FUNCTION_BLOCK OutputSender (* Composite Function Block Type *)
  (* Standard: 61499-2 *)
  (* Version 0.0, 6/20/2018, Rediska, nxtControl GmbH, template *)
  PACKAGE Main;
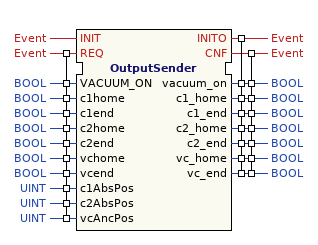
  EVENT_INPUT
    INIT; (* Initialization Request *)
    REQ WITH VACUUM_ON, c1home, c1end, c2home, c2end, vchome, vcend, c1AbsPos, c2AbsPos, vcAncPos; (* Normal Execution Request *)
  END_EVENT
  EVENT_OUTPUT
    INITO WITH vacuum_on, c1_home, c1_end, c2_home, c2_end, vc_home, vc_end; (* Initialization Confirm *)
    CNF WITH vacuum_on, c1_home, c1_end, c2_home, c2_end, vc_home, vc_end; (* Execution Confirmation *)
  END_EVENT
  VAR_INPUT
    VACUUM_ON : BOOL;
    c1home : BOOL;
    c1end : BOOL;
    c2home : BOOL;
    c2end : BOOL;
    vchome : BOOL;
    vcend : BOOL;
    c1AbsPos : UINT;
    c2AbsPos : UINT;
    vcAncPos : UINT;
  END_VAR
  VAR_OUTPUT
    vacuum_on : BOOL;
    c1_home : BOOL;
    c1_end : BOOL;
    c2_home : BOOL;
    c2_end : BOOL;
    vc_home : BOOL;
    vc_end : BOOL;
  END_VAR
  FBS
    FB2 : TCPIO(PORT := ;127.0.0.1:64998);
    FB3 : OutputDecompressor(delimiter := ;);
    FB1 : OutputCompressor(delimiter := ;, QI := TRUE);
  END_FBS
  EVENT_CONNECTIONS
    INIT TO FB1.INIT;
    REQ TO FB1.REQ;
    FB1.INITO TO FB2.INIT;
    FB1.CNF TO FB2.REQ;
    FB2.CNF TO FB2.ACK;
    FB2.INITO TO FB3.INIT;
    FB2.IND TO FB3.REQ;
    FB3.INITO TO INITO;
    FB3.CNF TO CNF;
  END_CONNECTIONS
  DATA_CONNECTIONS
    VACUUM_ON TO FB1.vacuum_on;
    c1home TO FB1.c1_home;
    c1end TO FB1.c1_end;
    c2home TO FB1.c2_home;
    c2end TO FB1.c2_end;
    vchome TO FB1.vc_home;
    vcend TO FB1.vc_end;
    FB1.QO TO FB2.QI;
    FB1.result TO FB2.DATAOUT;
    FB2.QO TO FB3.QI;
    FB2.DATAIN TO FB3.input;
    FB3.vacuum_on TO vacuum_on;
    FB3.c1_home TO c1_home;
    FB3.c1_end TO c1_end;
    FB3.c2_home TO c2_home;
    FB3.c2_end TO c2_end;
    FB3.vc_home TO vc_home;
    FB3.vc_end TO vc_end;
    c1AbsPos TO FB1.c1_abs_pos;
    c2AbsPos TO FB1.c2_abs_pos;
    vcAncPos TO FB1.vc_abs_pos;
  END_CONNECTIONS
END_FUNCTION_BLOCK
